(* 32-bit counter with count value as VAR_IN_OUT to allow count value to be set externally *)
FUNCTION_BLOCK FB_CTU32
VAR_INPUT
	bInput			: BOOL;		(* FALSE-TRUE increments counter value *)
	bReset			: BOOL;		(* set TRUE to reset counter value to 0 *)
	nThreshold		: UDINT;	(* threshold at which bOutput is set TRUE *)
END_VAR
VAR_IN_OUT
	nCounter		: UDINT;	(* counter value *)
END_VAR
VAR_OUTPUT
	bOutput			: BOOL;		(* nCounter >= nTheshold *)
END_VAR
VAR
	fbInputEdge		: R_TRIG;
END_VAR
(*
-------------------------------------------------------------------------------------------------
Date		Version	Author	Comments
-------------------------------------------------------------------------------------------------
30/01/2015	3.00.00	PB		No change

-------------------------------------------------------------------------------------------------
05/02/10	1.00.00	PB		Initial release

-------------------------------------------------------------------------------------------------
*)

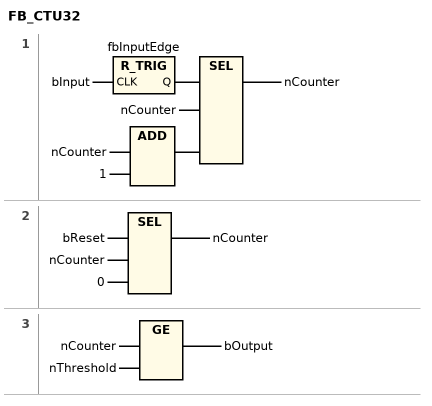
// NETWORK 1
fbInputEdge(CLK := bInput); // R_TRIG
nCounter := SEL(fbInputEdge.Q, nCounter, nCounter + 1);

// NETWORK 2
nCounter := SEL(bReset, nCounter, 0);

// NETWORK 3
bOutput := nCounter >= nThreshold;

END_FUNCTION_BLOCK

(* stored: Version 1.1.0.1, ProductVersion 3.1.4024.15
   POU FB_CTU32: Id {21ed98a5-7bac-4844-a87f-b23760c085d1}, SpecialFunc None *)
